Staubli VAL3: show_menu.pgx

program show_menu(screen& x_sScreen, num& x_nNum_choosed)
begin


  userPage(x_sScreen)
  title(x_sScreen,"Choose sub")

  gotoxy(x_sScreen,0,0)
  putln(x_sScreen,"F1)Filter 1 pick/bin")
  gotoxy(x_sScreen,0,1)
  putln(x_sScreen,"F2)Filter 2 pick/bin")
  gotoxy(x_sScreen,0,2)
  putln(x_sScreen,"F3)Filter 3 pick/bin")
  gotoxy(x_sScreen,0,3)
  putln(x_sScreen,"F4)Shelf pick/fixture (depreciated)")
  gotoxy(x_sScreen,0,4)
  putln(x_sScreen,"F5)Assemble")
  //---------------
  //  HRAS Lite
  //---------------
  gotoxy(x_sScreen,0,5)
  putln(x_sScreen,"F6)Cell to back secure f2f3")
  gotoxy(x_sScreen,0,6)
  putln(x_sScreen,"F7)Auto ver1")
  gotoxy(x_sScreen,0,7)
  putln(x_sScreen,"F8)Auto ver2 (multi")
  gotoxy(x_sScreen,0,8)
  putln(x_sScreen,"q)Cell to back secure f1f2f3")
  gotoxy(x_sScreen,0,9)
  putln(x_sScreen,"w)CAuto ver2 (single")

  //anykey
  x_nNum_choosed = get(x_sScreen)
  cls(x_sScreen)
end
